Staubli VAL3: socketRead.pgx

program socketRead()
begin
end
